// TIA Portal V20 export
TYPE "type_emRelations_em6_cmStatus"
// stored: Access Published, Namespace Unit1
   STRUCT
      HotpressLeftSafetyPin : "LBC_typeDigitalSignalControlNode";
      HotpressLeftJRDetect : "LBC_typeDigitalSignalControlNode";
      HotpressLeftStageLiftFrontUpDown : "LBC_typeTwoWayActuatorControlNode";
      HotpressLeftStageLiftRearUpDown : "LBC_typeTwoWayActuatorControlNode";
      HotpressLeftStageLiftAllUpDown : "LBC_typeTwoWayActuatorControlNode";
      HotPressLeftServoPress : "LER_typeServoPressControlNode";
      HotPressLeftTemperature : "LER_typeHeaterControlNode";
   END_STRUCT;
END_TYPE
